(*********************************** G.D S.p.A. - Technical Department ***********************************
============= PROGRAM INFO ============
FOLDER:             TBD
MACHINES INVOLVED:  TBD 

============= DESCRIPTION =============
csp - Upstream interface

============= REVISIONS ===============
Date		Version	 	Author      	Description             
----------	-------		------------  	--------------------------------------------
2019/10/07 	0000.00	 	W. Gerstner		Creation of the PRG

**********************************************************************************************************)
(*$R
	process_ref := prc;
$*)
PROGRAM csp_main_interface_upstream
VAR
	prc:					process;
	prc_path:				STRING;	

END_VAR

_read_var_input();

_object_manager();

IF NOT objects_running()
THEN
	RETURN;	
END_IF

_read_process_image();

_mode_manager();

CASE process_get_mode(prc) of
	MODE_ABSENT,
	MODE_INACTIVE:
		RETURN;
	MODE_TEST:
		_handle_process_test();
END_CASE

_set_runtime_properties();

(********************************* BODY *********************************)

(************************************************************************)

_handle_messages();

_write_output();

ACTION _handle_messages:
;
END_ACTION

ACTION _handle_process_test:
;
END_ACTION

ACTION _mode_manager:
IF process_mode_req_is_pending(prc)
THEN
    process_apply_mode_req_first_step(prc);
    CASE process_get_mode(prc) OF
        MODE_TO_ABSENT:
			;
        MODE_TO_INACTIVE:
			;
        MODE_TO_TEST:
			;
        MODE_TO_OPERATIONAL:
			;
    END_CASE
    process_apply_mode_req_second_step(prc);
END_IF
END_ACTION

ACTION _object_manager:
IF objects_initialization()
THEN
	sub_process_init(
		object_name					:= 'csp_main_interface_upstream.prc', 
		process						:= csp_main_interface.prc, 
		CONVERSION_this				:= prc);
		
	prc_path 						:= process_get_path(prc);
END_IF

IF objects_running()
THEN
	process_cycle(prc);
END_IF
END_ACTION

ACTION _read_process_image:
;
END_ACTION

ACTION _read_var_input:
;
END_ACTION

ACTION _set_runtime_properties:
;
END_ACTION

ACTION _write_output:
;
END_ACTION

END_PROGRAM

(* stored: Version 1.1.0.1, ProductVersion 3.1.4022.12
   POU csp_main_interface_upstream: Id {c288bedf-c8d1-40c5-ba3e-15c3008a59c4}, SpecialFunc None
   Action _handle_messages: Id {b367d570-b112-4ac1-ab37-c355de61b7bb}
   Action _handle_process_test: Id {08f63075-583d-4a8c-aae4-2398b63328ee}
   Action _mode_manager: Id {551bb96c-7f9f-4973-8878-c461cab255c0}
   Action _object_manager: Id {873f7dad-574e-43f6-89a2-feb1b982de8b}
   Action _read_process_image: Id {8ee8d8d4-71a6-45cd-bcd7-f6be564b0c00}
   Action _read_var_input: Id {7f07ccb9-1f2d-463c-903c-22bc34cf1b42}
   Action _set_runtime_properties: Id {beb0ad8c-9474-47f1-9956-4ed2d9bdd0f9}
   Action _write_output: Id {434c3c28-2885-41d0-bf33-b6b2f29ec723} *)
